{attribute 'qualified_only'}
{attribute 'strict'}
{attribute 'to_string'}
TYPE E_Axis :
(
	Disabled,
	Enabled,
	Idle,
	MoveAbs,
	Stop,
	Error,
	Reset,
	ManualMode
);
END_TYPE

(* stored: Version 1.1.0.1, ProductVersion 3.1.4024.9
   DUT E_Axis: Id {c10f7c7f-ed0d-4007-b87f-c6c078aa34a4} *)
